// TIA Portal V19 export
TYPE "MatCounterAlr"
// stored: Access Published
   STRUCT
      CounterNotInOperation : Bool;
   END_STRUCT;
END_TYPE
